(* IEC 61131-3 sources: repolevel_ST_code_completion/output/0122完整版本_无planner目前sota/repoeval_three-axis_CNC_motion/readful_result_no_provide, 4 files *)

(* ---- FB_TripleAxisHoming.st ---- *)
VAR
	fbHomingX			:	SMC_HOMING;			//X轴回零功能块
	fbHomingY			:	SMC_HOMING;			//Y轴回零功能块
	fbHomingZ			:	SMC_HOMING;			//Z轴回零功能块
	bXHomingDone		:	BOOL;				//X轴回零完成标志
	bYHomingDone		:	BOOL;				//Y轴回零完成标志
	bZHomingDone		:	BOOL;				//Z轴回零完成标志
	bXHomingError		:	BOOL;				//X轴回零错误标志
	bYHomingError		:	BOOL;				//Y轴回零错误标志
	bZHomingError		:	BOOL;				//Z轴回零错误标志
	sTempErrorString	:	STRING;				//临时错误信息字符串
END_VAR

IF bExecute THEN
	bBusy := TRUE;
	bError := FALSE;
	sErrorString := '';

	// X轴回零过程
	fbHomingX.Axis := AxisX;
	fbHomingX.Execute := NOT bXHomingDone;
	fbHomingX.Velocity := fVelocityFast;
	fbHomingX.Acceleration := fAcceleration;
	fbHomingX.Deceleration := fDeceleration;
	fbHomingX.HomeSwitch := bAxisXRefSwitch;
	fbHomingX();
	bXHomingDone := fbHomingX.Done;
	bXHomingError := fbHomingX.Error;

	// Y轴回零过程
	fbHomingY.Axis := AxisY;
	fbHomingY.Execute := NOT bYHomingDone AND bXHomingDone;
	fbHomingY.Velocity := fVelocityFast;
	fbHomingY.Acceleration := fAcceleration;
	fbHomingY.Deceleration := fDeceleration;
	fbHomingY.HomeSwitch := bAxisYRefSwitch;
	fbHomingY();
	bYHomingDone := fbHomingY.Done;
	bYHomingError := fbHomingY.Error;

	// Z轴回零过程
	fbHomingZ.Axis := AxisZ;
	fbHomingZ.Execute := NOT bZHomingDone AND bYHomingDone;
	fbHomingZ.Velocity := fVelocityFast;
	fbHomingZ.Acceleration := fAcceleration;
	fbHomingZ.Deceleration := fDeceleration;
	fbHomingZ.HomeSwitch := bAxisZRefSwitch;
	fbHomingZ();
	bZHomingDone := fbHomingZ.Done;
	bZHomingError := fbHomingZ.Error;

	// 错误处理
	IF bXHomingError THEN
		bError := TRUE;
		sTempErrorString := fbHomingX.ErrorID;
	ELSIF bYHomingError THEN
		bError := TRUE;
		sTempErrorString := fbHomingY.ErrorID;
	ELSIF bZHomingError THEN
		bError := TRUE;
		sTempErrorString := fbHomingZ.ErrorID;
	END_IF;

	IF bError THEN
		sErrorString := CONCAT('Homing Error: ', sTempErrorString);
		bBusy := FALSE;
		RETURN;
	END_IF;

	// 回零完成状态
	bAxisXHomeOK := bXHomingDone;
	bAxisYHomeOK := bYHomingDone;
	bAxisZHomeOK := bZHomingDone;
	bHomeOK := bXHomingDone AND bYHomingDone AND bZHomingDone;

	IF bHomeOK THEN
		bBusy := FALSE;
	END_IF;
ELSE
	bBusy := FALSE;
	bHomeOK := FALSE;
	bAxisXHomeOK := FALSE;
	bAxisYHomeOK := FALSE;
	bAxisZHomeOK := FALSE;
	bError := FALSE;
	sErrorString := '';
END_IF;
END_FUNCTION_BLOCK

(* ---- FB_TripleAxisPower.st ---- *)
VAR
	fbPowerX		:	MC_POWER;			//X轴电源控制
	fbPowerY		:	MC_POWER;			//Y轴电源控制
	fbPowerZ		:	MC_POWER;			//Z轴电源控制
	bErrorX			:	BOOL;				//X轴错误标志
	bErrorY			:	BOOL;				//Y轴错误标志
	bErrorZ			:	BOOL;				//Z轴错误标志
	sErrorX			:	STRING;				//X轴错误信息
	sErrorY			:	STRING;				//Y轴错误信息
	sErrorZ			:	STRING;				//Z轴错误信息
END_VAR

fbPowerX(
	Enable := bServoEnable,
	bRegulatorOn := bServoEnable,
	bDriveStart := bServoEnable,
	Axis := AxisX
);

fbPowerY(
	Enable := bServoEnable,
	bRegulatorOn := bServoEnable,
	bDriveStart := bServoEnable,
	Axis := AxisY
);

fbPowerZ(
	Enable := bServoEnable,
	bRegulatorOn := bServoEnable,
	bDriveStart := bServoEnable,
	Axis := AxisZ
);

bAxisXReady := fbPowerX.Status = MC_POWER_STATUS.PowerOn;
bAxisYReady := fbPowerY.Status = MC_POWER_STATUS.PowerOn;
bAxisZReady := fbPowerZ.Status = MC_POWER_STATUS.PowerOn;

bErrorX := fbPowerX.Error;
bErrorY := fbPowerY.Error;
bErrorZ := fbPowerZ.Error;

sErrorX := fbPowerX.ErrorID;
sErrorY := fbPowerY.ErrorID;
sErrorZ := fbPowerZ.ErrorID;

bError := bErrorX OR bErrorY OR bErrorZ;

IF bError THEN
	IF bErrorX THEN
		sErrorString := 'X Axis Error: ' + sErrorX;
	ELSIF bErrorY THEN
		sErrorString := 'Y Axis Error: ' + sErrorY;
	ELSIF bErrorZ THEN
		sErrorString := 'Z Axis Error: ' + sErrorZ;
	END_IF;
ELSE
	sErrorString := '';
END_IF;

bReady := bAxisXReady AND bAxisYReady AND bAxisZReady;
END_FUNCTION_BLOCK

(* ---- FB_TripleAxisStop.st ---- *)
VAR
	fbStopX			:	MC_STOP;			//X轴停止
	fbStopY			:	MC_STOP;			//Y轴停止
	fbStopZ			:	MC_STOP;			//Z轴停止
	bStopXDone		:	BOOL;				//X轴停止完成
	bStopYDone		:	BOOL;				//Y轴停止完成
	bStopZDone		:	BOOL;				//Z轴停止完成
	bStopXError		:	BOOL;				//X轴停止错误
	bStopYError		:	BOOL;				//Y轴停止错误
	bStopZError		:	BOOL;				//Z轴停止错误
	sStopXErrorString:	STRING;				//X轴错误信息
	sStopYErrorString:	STRING;				//Y轴错误信息
	sStopZErrorString:	STRING;				//Z轴错误信息
END_VAR

fbStopX(
	Execute := bExecute,
	Deceleration := rDeceleration,
	Axis := AxisX
);
bStopXDone := fbStopX.Done;
bStopXError := fbStopX.Error;
sStopXErrorString := fbStopX.ErrorID;

fbStopY(
	Execute := bExecute,
	Deceleration := rDeceleration,
	Axis := AxisY
);
bStopYDone := fbStopY.Done;
bStopYError := fbStopY.Error;
sStopYErrorString := fbStopY.ErrorID;

fbStopZ(
	Execute := bExecute,
	Deceleration := rDeceleration,
	Axis := AxisZ
);
bStopZDone := fbStopZ.Done;
bStopZError := fbStopZ.Error;
sStopZErrorString := fbStopZ.ErrorID;

bDone := bStopXDone AND bStopYDone AND bStopZDone;
bBusy := NOT bDone;
bError := bStopXError OR bStopYError OR bStopZError;

IF bStopXError THEN
	sErrorString := sStopXErrorString;
ELSIF bStopYError THEN
	sErrorString := sStopYErrorString;
ELSIF bStopZError THEN
	sErrorString := sStopZErrorString;
ELSE
	sErrorString := '';
END_IF;
END_FUNCTION_BLOCK

(* ---- INIT_CNC_System.st ---- *)
VAR
    bInitSuccess : BOOL;
END_VAR

fbSMC_ReadNCFile(bExecute := FALSE);
fbSMC_NCDecoder(bExecute := FALSE, ncprog := fbSMC_ReadNCFile.ncprog);
fbSMC_CheckVelocities(bExecute := FALSE);
fbSMC_Interpolator(bExecute := FALSE);

fbSMC_AXISX_HOMING(bExecute := FALSE, Axis := AxisX);
fbSMC_AXISY_HOMING(bExecute := FALSE, Axis := AxisY);
fbSMC_AXISZ_HOMING(bExecute := FALSE, Axis := AxisZ);

fbMC_AXISX_STOP(bExecute := FALSE, Axis := AxisX);
fbMC_AXISY_STOP(bExecute := FALSE, Axis := AxisY);
fbMC_AXISZ_STOP(bExecute := FALSE, Axis := AxisZ);

bInitSuccess := TRUE;
RETURN bInitSuccess;
END_FUNCTION
